PROGRAM ScanBuffer
VAR
	// Default
	Done: BOOL;
	
	// Goto Buffer id
	BufferId: INT;
	BufferIdReady: BOOL;
	
	// Invalid Buffer part
	InvalidPart: BOOL;
	Quatity: INT;
END_VAR

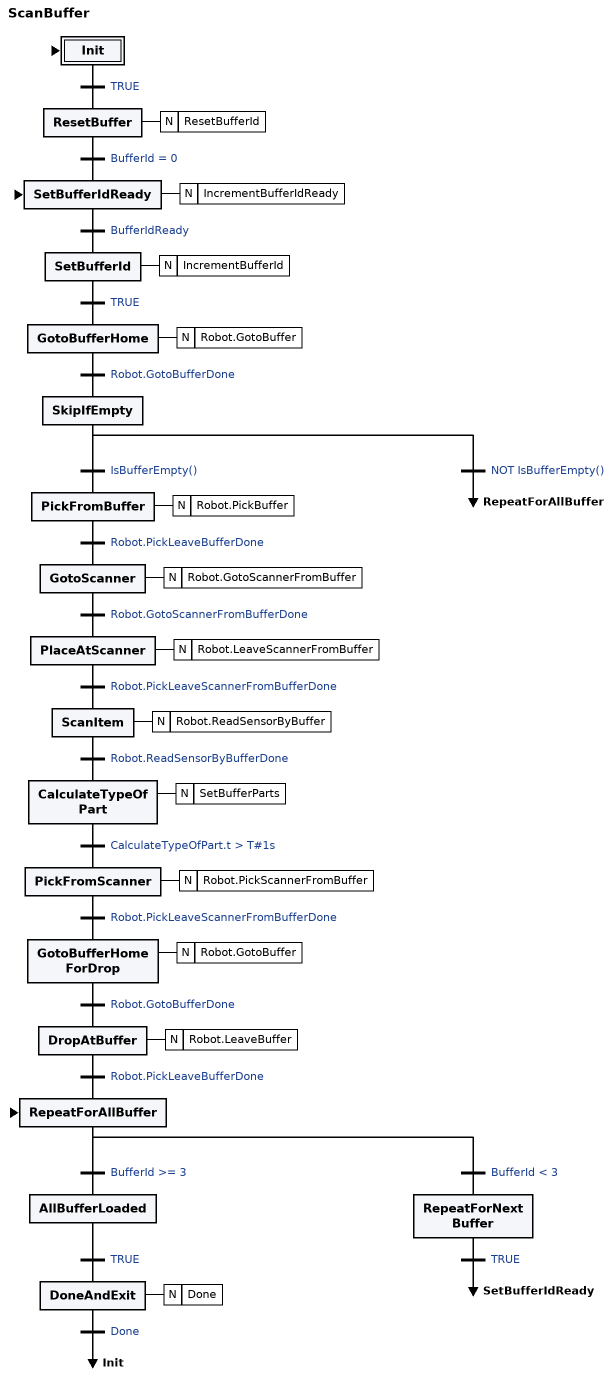
INITIAL_STEP Init:
END_STEP
TRANSITION FROM Init TO ResetBuffer
    := TRUE;
END_TRANSITION
STEP ResetBuffer:
    ResetBufferId(N);
END_STEP
TRANSITION FROM ResetBuffer TO SetBufferIdReady
    := BufferId = 0;
END_TRANSITION
STEP SetBufferIdReady:
    IncrementBufferIdReady(N);
END_STEP
TRANSITION FROM SetBufferIdReady TO SetBufferId
    := BufferIdReady;
END_TRANSITION
STEP SetBufferId:
    IncrementBufferId(N);
END_STEP
TRANSITION FROM SetBufferId TO GotoBufferHome
    := TRUE;
END_TRANSITION
STEP GotoBufferHome:
    Robot.GotoBuffer(N);
END_STEP
TRANSITION FROM GotoBufferHome TO SkipIfEmpty
    := Robot.GotoBufferDone;
END_TRANSITION
STEP SkipIfEmpty:
END_STEP
TRANSITION FROM SkipIfEmpty TO PickFromBuffer
    := IsBufferEmpty();
END_TRANSITION
TRANSITION FROM SkipIfEmpty TO RepeatForAllBuffer
    := NOT IsBufferEmpty();
END_TRANSITION
STEP PickFromBuffer:
    Robot.PickBuffer(N);
END_STEP
TRANSITION FROM PickFromBuffer TO GotoScanner
    := Robot.PickLeaveBufferDone;
END_TRANSITION
STEP GotoScanner:
    Robot.GotoScannerFromBuffer(N);
END_STEP
TRANSITION FROM GotoScanner TO PlaceAtScanner
    := Robot.GotoScannerFromBufferDone;
END_TRANSITION
STEP PlaceAtScanner:
    Robot.LeaveScannerFromBuffer(N);
END_STEP
TRANSITION FROM PlaceAtScanner TO ScanItem
    := Robot.PickLeaveScannerFromBufferDone;
END_TRANSITION
STEP ScanItem:
    Robot.ReadSensorByBuffer(N);
END_STEP
TRANSITION FROM ScanItem TO CalculateTypeOfPart
    := Robot.ReadSensorByBufferDone;
END_TRANSITION
STEP CalculateTypeOfPart:
    SetBufferParts(N);
END_STEP
TRANSITION FROM CalculateTypeOfPart TO PickFromScanner
    := CalculateTypeOfPart.t > T#1s;
END_TRANSITION
STEP PickFromScanner:
    Robot.PickScannerFromBuffer(N);
END_STEP
TRANSITION FROM PickFromScanner TO GotoBufferHomeForDrop
    := Robot.PickLeaveScannerFromBufferDone;
END_TRANSITION
STEP GotoBufferHomeForDrop:
    Robot.GotoBuffer(N);
END_STEP
TRANSITION FROM GotoBufferHomeForDrop TO DropAtBuffer
    := Robot.GotoBufferDone;
END_TRANSITION
STEP DropAtBuffer:
    Robot.LeaveBuffer(N);
END_STEP
TRANSITION FROM DropAtBuffer TO RepeatForAllBuffer
    := Robot.PickLeaveBufferDone;
END_TRANSITION
STEP RepeatForAllBuffer:
END_STEP
TRANSITION FROM RepeatForAllBuffer TO AllBufferLoaded
    := BufferId >= 3;
END_TRANSITION
STEP AllBufferLoaded:
END_STEP
TRANSITION FROM AllBufferLoaded TO DoneAndExit
    := TRUE;
END_TRANSITION
TRANSITION FROM RepeatForAllBuffer TO RepeatForNextBuffer
    := BufferId < 3;
END_TRANSITION
STEP RepeatForNextBuffer:
END_STEP
TRANSITION FROM RepeatForNextBuffer TO SetBufferIdReady
    := TRUE;
END_TRANSITION
STEP DoneAndExit:
    Done(N);
END_STEP
TRANSITION FROM DoneAndExit TO Init
    := Done;
END_TRANSITION

ACTION IncrementBufferId:
IF BufferIdReady = TRUE THEN
	BufferId := BufferId + 1;
	BufferIdReady := FALSE;
END_IF
END_ACTION

ACTION IncrementBufferIdReady:
BufferIdReady := TRUE;
END_ACTION

METHOD IsBufferEmpty : BOOL
VAR_INPUT
END_VAR
CASE BufferId OF
	1:
		IF GVL.BufferProducts.Storage1.Quatity > 0 THEN
			IsBufferEmpty := FALSE;
		ELSE
			IsBufferEmpty := TRUE;
		END_IF
	2:
		IF GVL.BufferProducts.Storage2.Quatity > 0 THEN
			IsBufferEmpty := FALSE;
		ELSE
			IsBufferEmpty := TRUE;
		END_IF
	3:
		IF GVL.BufferProducts.Storage3.Quatity > 0 THEN
			IsBufferEmpty := FALSE;
		ELSE
			IsBufferEmpty := TRUE;
		END_IF
END_CASE
END_METHOD

ACTION ResetBufferId:
BufferId := 0;
END_ACTION

ACTION SetBufferParts:
IF Robot.IdentifyPartFB.Product = 'PLATE' THEN
	Quatity := 2;
ELSIF Robot.IdentifyPartFB.Product = 'CYLINDER' THEN
	Quatity := 4;
ELSIF Robot.IdentifyPartFB.Product = 'OCTAGON' THEN
	Quatity := 4;
ELSE
	Quatity := 0;
	GVL.mwStationStatus := 1000;
	
END_IF

CASE BufferId OF
	1:
		GVL.BufferProducts.Storage1.Quatity := Quatity;
		GVL.BufferProducts.Storage1.Component := Robot.IdentifyPartFB.Component;
	2:
		GVL.BufferProducts.Storage2.Quatity := Quatity;
		GVL.BufferProducts.Storage2.Component := Robot.IdentifyPartFB.Component;
	3:
		GVL.BufferProducts.Storage3.Quatity := Quatity;
		GVL.BufferProducts.Storage3.Component := Robot.IdentifyPartFB.Component;
END_CASE
END_ACTION

ACTION SkipScan:
GVL.BufferProducts.Storage1.Component := 'REDPLATE';
GVL.BufferProducts.Storage1.Quatity := 2;
GVL.BufferProducts.Storage2.Component := 'REDCYLINDER';
GVL.BufferProducts.Storage2.Quatity := 4;
GVL.BufferProducts.Storage3.Component := 'REDOCTAGON';
GVL.BufferProducts.Storage3.Quatity := 4;
END_ACTION

END_PROGRAM

(* stored: Version 1.1.0.1, ProductVersion 3.1.4024.12
   POU ScanBuffer: Id {b9ec7242-378c-418b-8ad6-f7b7e8aacb8b}, SpecialFunc None
   Action IncrementBufferId: Id {46e1d539-82e0-4ce6-b13d-a1b27ef0a3ae}
   Action IncrementBufferIdReady: Id {e5cee1d1-a31a-4e44-8aae-2f9ae6bd3984}
   Method IsBufferEmpty: Id {21e30fd4-0dfb-4559-8133-60a9d4128c97}
   Action ResetBufferId: Id {92328b5d-044c-405c-be31-2c2a56150132}
   Action SetBufferParts: Id {3202afd0-f2f5-4384-9608-1ea0c3f2d82c}
   Action SkipScan: Id {815b63ae-bd7d-462e-839c-fccc2273b0b3} *)
